Omron CX-Programmer project NewProject (CX-Programmer 9.80)

# PLC NewPLC1: CP1L M

## Global symbols (name address type ; comment)
W0.00 BOOL  ; cond_marche_motuer_courroie

## Program NewProgram1 (cyclic task 0)
Local symbols
Cap_ind_courroie_haut 0.02 BOOL  ; Cap. ind. courroie haut
Cap_indi_courroie_bas 0.03 BOOL  ; Cap. ind. courroie bas
M_Rouleaux_table_fix 100.03 BOOL  ; M_Rouleaux_table_fix
M_courroie 100.00 BOOL  ; motuer courroie
M_elev_courroie 100.02 BOOL  ; M_elev_courroie
Montée_compensateur 100.01 BOOL  ; Montée_compensateur
PH_entree_rangée 0.00 BOOL  ; FC_entree_rangée
PH_présence_rangée_fin_table_fixe 0.05 BOOL  ; PH_présence_rangée_fin_table_fixe
PH_rangée_sur_table 0.01 BOOL  ; PH_rangée_sur_table
State_moteur_courroie H0.00 BOOL  ; 1=run 0=stop
cap_comp_pas_a_pas 0.08 BOOL  ; cap_comp_pas_a_pas
cap_compensateur_bas 0.07 BOOL  ; cap.compensateur_haut
cap_compensateur_haut 0.06 BOOL  ; cap.compensateur_haut
cond_marche_moteur_courroie W0.00 BOOL  ; cond_marche_moteur_courroie
cond_moteur_elev_courroie W0.01 BOOL  ; cond_moteur_elev_courroie
condition_Montée_compensateur W0.02 BOOL  ; condition_Montée_compensateur
condition_descent_compensateur W0.04 BOOL  ; condition_descent_compensateur
condition_moteur_rouleaux_Table_fix W0.03 BOOL  ; condition_moteur_rouleaux_table_fix
descent_compensateur 100.04 BOOL  ; descent_compensateur
rangée_sur_compensateur 0.04 BOOL  ; rangée_sur_compensateur
state_descent_courroie H1.00 BOOL  ; descent=1 Stop=0
state_montée_courroie H1.01 BOOL  ; montée=1 stop =0

### Section system_moteur_courroie

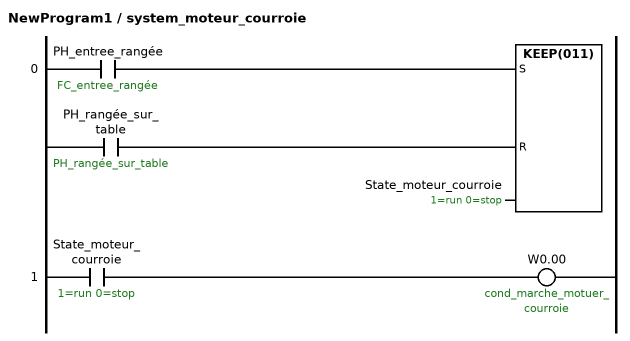
; rung 0
LD PH_entree_rangée  ; FC_entree_rangée
LD PH_rangée_sur_table  ; PH_rangée_sur_table
KEEP(011) State_moteur_courroie  ; 1=run 0=stop
; rung 1
LD State_moteur_courroie  ; 1=run 0=stop
OUT W0.00  ; cond_marche_motuer_courroie

### Section elevateur_courroie

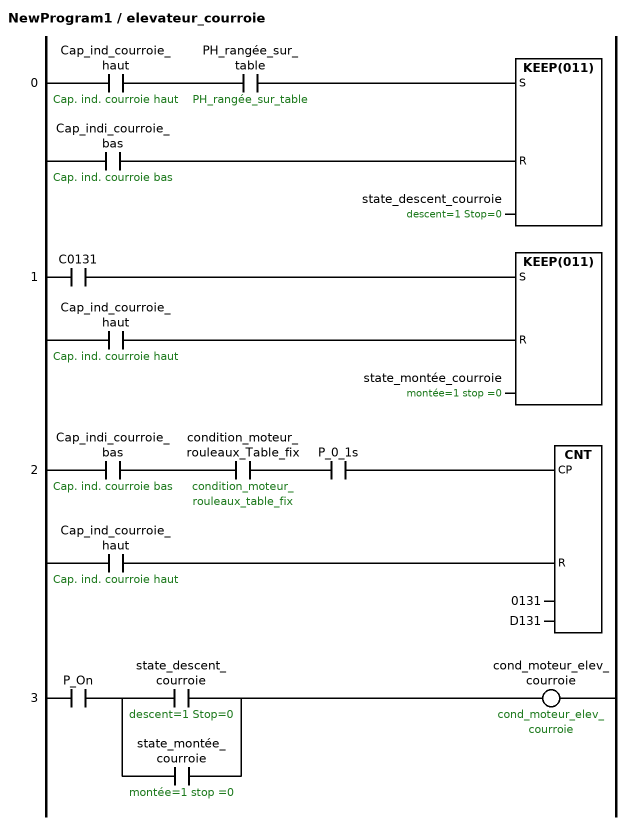
; rung 0
LD Cap_ind_courroie_haut  ; Cap. ind. courroie haut
AND PH_rangée_sur_table  ; PH_rangée_sur_table
LD Cap_indi_courroie_bas  ; Cap. ind. courroie bas
KEEP(011) state_descent_courroie  ; descent=1 Stop=0
; rung 1
LD C0131
LD Cap_ind_courroie_haut  ; Cap. ind. courroie haut
KEEP(011) state_montée_courroie  ; montée=1 stop =0
; rung 2
LD Cap_indi_courroie_bas  ; Cap. ind. courroie bas
AND condition_moteur_rouleaux_Table_fix  ; condition_moteur_rouleaux_table_fix
AND P_0_1s
LD Cap_ind_courroie_haut  ; Cap. ind. courroie haut
CNT 0131 D131
; rung 3
LD P_On
LD state_descent_courroie  ; descent=1 Stop=0
OR state_montée_courroie  ; montée=1 stop =0
ANDLD
OUT cond_moteur_elev_courroie  ; cond_moteur_elev_courroie

### Section compensateur

### Section table_mobile

### Section output

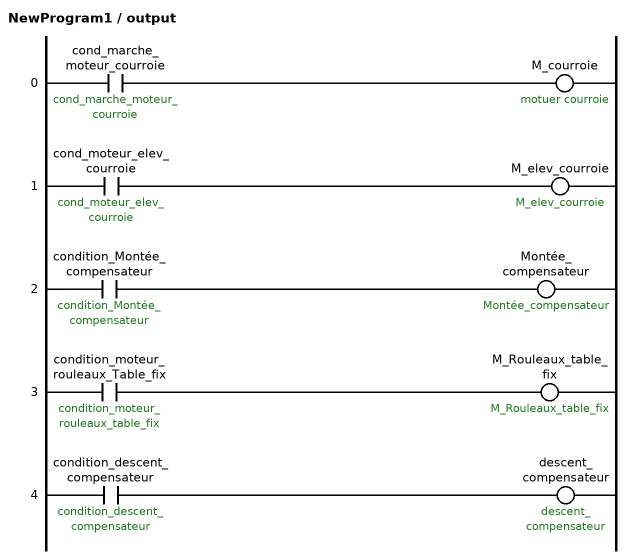
; rung 0
LD cond_marche_moteur_courroie  ; cond_marche_moteur_courroie
OUT M_courroie  ; motuer courroie
; rung 1
LD cond_moteur_elev_courroie  ; cond_moteur_elev_courroie
OUT M_elev_courroie  ; M_elev_courroie
; rung 2
LD condition_Montée_compensateur  ; condition_Montée_compensateur
OUT Montée_compensateur  ; Montée_compensateur
; rung 3
LD condition_moteur_rouleaux_Table_fix  ; condition_moteur_rouleaux_table_fix
OUT M_Rouleaux_table_fix  ; M_Rouleaux_table_fix
; rung 4
LD condition_descent_compensateur  ; condition_descent_compensateur
OUT descent_compensateur  ; descent_compensateur

### Section END
; rung 0
END(001)